FUNCTION_BLOCK FB_Utilities_Control_Old
VAR_INPUT
	i_init_utilities 		: BOOL;
	i_activate_util			: BOOL;
	i_shutdown_utilities 	: BOOL;
	i_fault_reset			: BOOL;
	
	i_state_req				: INT;
	
	i_cooling_pump_req		: ST_Util_Service_Req;
	i_deadair_pump_req		: ST_Util_Service_Req;
	i_steam_system_req		: ST_Util_Service_Req;
	i_purge_assist_req		: ST_Util_Service_Req;
END_VAR
VAR_OUTPUT
	o_bop_error				: BOOL;
	o_bop_warmup_sts		: ST_SeqSts;
	o_bop_activate_sts		: ST_SeqSts;
	o_bop_shutdown_sts		: ST_SeqSts;
END_VAR
VAR
	in_bop_warmup_sts 		AT %I* : BYTE;
	in_bop_activate_sts		AT %I* : BYTE;
	in_bop_shutdown_sts		AT %I* : BYTE;
	in_bop_error_sts		AT %I* : BOOL;
	in_bop_error_code		AT %I* : DWORD;
	
	comms_fault		: BOOL;
	
	out_util_state_req 		AT %Q* : INT; // 0 = Idle, 1 = warmup, 2 = activavte, 3 = shutdown 
	out_util_reset_fault	AT %Q* : BOOL;
	
	
	
	cooling_pump	: FB_Utilities_Service;
	dead_air_pump	: FB_Utilities_Service;
	steam_sytem 	: FB_Utilities_Service;
	purge_assist 	: FB_Utilities_Service;
	
	//util_dispatcher	: FB_Utilities_Dispatcher;
	
	cooling_pump_dispatch : FB_Service_Dispatcher();
	deadair_pump_dispatch : FB_Service_Dispatcher();
	
	util_state : ( Idle := 0, Warmup := 1, Activate := 2, Shutdown := 3, Error) ;
	
	cooling_pump_req : ST_Util_Service_Req;
	
	cooling_pump_set_output : FB_SetOutput;
	
END_VAR

PROPERTY CoolingPump_Assigned_RS :
GET
CoolingPump_Assigned_RS := cooling_pump_dispatch.o_assigned_rs_number;
END_GET
END_PROPERTY

METHOD CoolingPump_Control : BOOL
VAR_INPUT
END_VAR
VAR
	service_req : REAL;
END_VAR
// Clear Queue if pump is faulted from utilities controller
IF NOT cooling_pump.o_service_sts.faulted AND NOT comms_fault AND  HMI.util_auto_mode THEN 
	cooling_pump_req := i_cooling_pump_req;
ELSE
	cooling_pump_dispatch.Clear_Queue();
END_IF


// manage the cooling pump assignmnet queue based on request form reactor set controller
cooling_pump_dispatch( i_service_req := i_cooling_pump_req, i_shared_rs_count := 8, i_rs_module_constrain := FALSE);


IF hmi.util_auto_mode THEN 
	// set  the cooling pump on/off command based on dispacher assignnments
	IF cooling_pump_dispatch.o_service_req THEN 
		service_req := E_Util_Service_Req.On;
	ELSE
		service_req := E_Util_Service_Req.Off;
	END_IF	
END_IF


IF ( i_cooling_pump_req.request_cmd = E_Util_Service_Req.Reset OR hmi.util_cooling_pump_cmd = E_Util_Service_Req.Reset) AND cooling_pump.o_service_sts.faulted THEN 
		service_req := i_cooling_pump_req.request_cmd;
	END_IF

	
 cooling_pump_set_output(io_in1 := service_req, io_in2 := hmi.util_cooling_pump_cmd); 	
 cooling_pump.i_service_req.request_cmd := TO_INT(cooling_pump_set_output.o_set_value);	
	
//  cooling pump ios ( cmd + sts )  mapping to/from utilities controller 
cooling_pump();
END_METHOD

PROPERTY CoolingPump_Sts : ST_Util_Service_Sts
GET
CoolingPump_Sts := cooling_pump.o_service_sts;
END_GET
END_PROPERTY

METHOD DeadAirPump_Control : BOOL
VAR_INPUT
END_VAR

deadair_pump_dispatch( i_service_req := i_deadair_pump_req);
dead_air_pump();
END_METHOD

PROPERTY DeadAirPump_Sts : ST_Util_Service_Sts
GET
DeadAirPump_Sts := dead_air_pump.o_service_sts;
END_GET
END_PROPERTY

METHOD GetSet_BOP_IOs : BOOL
VAR_INPUT
END_VAR

// Get IOs

F_Get_Seq_Status( i_seq_sts := in_bop_warmup_sts, o_seq_sts => o_bop_warmup_sts);
F_Get_Seq_Status( i_seq_sts := in_bop_activate_sts, o_seq_sts => o_bop_activate_sts);
F_Get_Seq_Status( i_seq_sts := in_bop_shutdown_sts, o_seq_sts => o_bop_shutdown_sts);

o_bop_error := in_bop_error_sts;
END_METHOD

PROPERTY PurgeAssist_Sts : ST_Util_Service_Sts
GET
PurgeAssist_Sts := purge_assist.o_service_sts;
END_GET
END_PROPERTY

METHOD State_Machine : BOOL
VAR_INPUT
END_VAR
IF i_state_req = E_Util_State_Cmd.Shutdown THEN
	util_state := Shutdown;
END_IF

CASE util_state OF 
	
	Idle : 
		IF i_state_req = E_Util_State_Cmd.Warmup  AND NOT in_bop_error_sts THEN 
			util_state := Warmup;
		ELSIF 	in_bop_error_sts THEN 
			util_state := Error;
		END_IF
	Warmup: 
		out_util_state_req := Warmup;
		IF NOT o_bop_warmup_sts.error THEN 
			IF o_bop_warmup_sts.completed AND i_state_req = E_Util_State_Cmd.Activate THEN 
				util_state := Activate;
			END_IF
		ELSE
			util_state := Error;
		END_IF
	Activate: 
		out_util_state_req := Activate;
		IF  o_bop_activate_sts.error THEN 
			util_state := Error;
		END_IF
		
	Shutdown : 
		out_util_state_req := Shutdown;
		IF NOT o_bop_shutdown_sts.error THEN 
			IF o_bop_shutdown_sts.completed THEN 
				util_state := Idle;
			END_IF
		ELSE
			util_state := Error;
		END_IF
	Error: 
		IF i_fault_reset THEN 
			out_util_reset_fault := TRUE;
			IF NOT in_bop_error_sts THEN
				util_state := Idle;
			END_IF
		END_IF
		
END_CASE
END_METHOD

PROPERTY SteamSystem_Sts : ST_Util_Service_Sts
GET
SteamSystem_Sts := steam_sytem.o_service_sts;
END_GET
END_PROPERTY

END_FUNCTION_BLOCK

(* stored: Version 1.1.0.1, ProductVersion 3.1.4024.12
   POU FB_Utilities_Control_Old: Id {8c6b6cdd-7265-4a56-a4b4-c8746bfbe857}, SpecialFunc None
   Property CoolingPump_Assigned_RS: Id {779fbffc-5bb8-48f2-a000-685aa64d8599}
   Get Get: Id {0e27d998-d7ce-4e5d-b03a-a81813c6f904}
   Method CoolingPump_Control: Id {87b36801-af68-47a8-9110-d4009490d768}
   Property CoolingPump_Sts: Id {7316fd9b-3061-4fa0-a714-ac480e11acfa}
   Get Get: Id {d3c6616e-43cf-48e4-87e3-0a629123ca49}
   Method DeadAirPump_Control: Id {2dddd7cc-b65c-4e22-bf02-7de4b30df3b7}
   Property DeadAirPump_Sts: Id {f06135dc-afa2-4efa-8940-c4c64349210e}
   Get Get: Id {38a46abb-2a3d-4082-898e-ce5b5951812b}
   Method GetSet_BOP_IOs: Id {26c09f7b-23c0-42f9-85d2-289bbda01008}
   Property PurgeAssist_Sts: Id {38bed4f6-0484-45ef-98fa-176288db34d8}
   Get Get: Id {77e09263-3af6-4d99-bf48-816409fdbc74}
   Method State_Machine: Id {098dda64-0e68-4a64-9b10-f955bc143fbc}
   Property SteamSystem_Sts: Id {db5902fe-8d31-4065-af95-3ebb7e1438d6}
   Get Get: Id {2452a151-60c9-4b17-ba95-54f6bd2be5a7} *)
